PROGRAM MAIN
VAR
END_VAR

END_PROGRAM

(* stored: Version 1.1.0.1
   POU MAIN: Id {70437695-90d8-427e-a4a4-ac80a32edb61} *)
